// TIA Portal project "First" (V17)

(* hardware
DEVICE "S7-400 station_1"  S7-400 station
   slot 0: "UR1_0"  UR1  6ES7 400-1TA01-0AA0
   slot 1: "PS 407 10A_1"  PS 407 10A  6ES7 407-0KA02-0AA0
   slot 3: "6ES7"  Unspecific CPU S7 400  6ES7 4XX-XXXXX-XXXX
   slot 4: "CP 443-1_1"  CP 443-1  6GK7 443-1EX11-0XE0  V2.7
*)

// ===== PLC "6ES7"  Unspecific CPU S7 400 =====

ORGANIZATION_BLOCK "Main"   // OB1, LAD
TITLE = "Main Program Sweep (Cycle)"
{ S7_Optimized_Access := 'FALSE' }
VERSION : 0.1
   VAR_TEMP
      OB1_EV_CLASS : Byte;   // Bits 0-3 = 1 (Coming event), Bits 4-7 = 1 (Event class 1)
      OB1_SCAN_1 : Byte;   // 1 (Cold restart scan 1 of OB 1), 3 (Scan 2-n of OB 1)
      OB1_PRIORITY : Byte;   // Priority of OB Execution
      OB1_OB_NUMBR : Byte;   // 1 (Organization block 1, OB1)
      OB1_RESERVED_1 : Byte;   // Reserved for system
      OB1_RESERVED_2 : Byte;   // Reserved for system
      OB1_PREV_CYCLE : Int;   // Cycle time of previous OB1 scan (milliseconds)
      OB1_MIN_CYCLE : Int;   // Minimum cycle time of OB1 (milliseconds)
      OB1_MAX_CYCLE : Int;   // Maximum cycle time of OB1 (milliseconds)
      OB1_DATE_TIME : Date_And_Time;   // Date and time OB1 started
   END_VAR
BEGIN
END_ORGANIZATION_BLOCK